// TwinCAT 3 PLC project TcoElements
// Title: TcoElements
// Company: Vortex.Library
// ProjectVersion: 0.6.0.913
// ProgramVersion: 3.1.4026.12
// libraries:
//   Tc2_Standard, * (Beckhoff Automation GmbH)
//   Tc2_System, * (Beckhoff Automation GmbH)
//   Tc3_Module, * (Beckhoff Automation GmbH)
//   TcoCore, 0.6.0.913 (Vortex.Library)
//   TcoUtilities, 0.6.0.913 (Vortex.Library)
// project tree:
//   Analog/TcoAi/ TcoAiAny.TcPOU (not stored), TcoAi.TcPOU (not stored), TcoAiConfig.TcDUT (not stored), TcoAiStatus.TcDUT (not stored)
//   Analog/TcoAo/ TcoAoConfig.TcDUT (not stored), TcoAoStatus.TcDUT (not stored), TcoAo.TcPOU (not stored)
//   Carousel/Base/ TcoCarouselBase.TcPOU (not stored)
//   Carousel/Structs/ eTcoCarouselDirection.TcDUT (not stored), TcoCarouselConfig.TcDUT (not stored), TcoCarouselStatus.TcDUT (not stored)
//   Carousel/Tasks/ TcoTurnTableTask.TcPOU (not stored)
//   Carousel/ TcoCarousel.TcPOU
//   Digital/TcoDi/ TcoDi.TcPOU, TcoDiConfig.TcDUT
//   Digital/TcoDo/ TcoDo.TcPOU
//   / PlcTask.TcTTO (not stored)
//   POUs/ MAIN.TcPOU (not stored)
// real-time tasks:
//   TASK PlcTask: cycle T#10ms, priority 20, ADS port 350
//   TASK PlcTask1: cycle T#10ms, priority 21, ADS port 351

// ---- Digital/TcoDi/TcoDiConfig.TcDUT
TYPE TcoDiConfig :
STRUCT
	IsFalseTimeOut : TIME := T#10S;
	IsTrueTimeOut : TIME := T#10S;
END_STRUCT
END_TYPE

// ---- Carousel/TcoCarousel.TcPOU
{attribute addProperty _turnTableName "<#Turn#>"}
{attribute addProperty _restoreName "<#Restore#>"}
FUNCTION_BLOCK TcoCarousel EXTENDS TcoCarouselBase
VAR_INPUT
		(*~
		<docu>
			<summary>
				This condition prevents the rotation of the table, possibly due to collisions with cylinders, axes, or other objects.
				Do not use signal from Light Curtain here.
			</summary>	
		</docu>
	~*)
	inSafetyCondition:BOOL;
	(*~
		<docu>
			<summary>
				The coded bites are stored in this word, which is valid for the base position of the carousel.
			</summary>	
		</docu>
	~*)
	inBasePositionNumber:WORD;
	
END_VAR
VAR
    {attribute addProperty Name "|[[1]Attribute_turnTableName]|"}
    _turnTask : TcoTurnTableTask(THIS^);

    {attribute addProperty Name "|[[1]Attribute_restoreName]|"}
    _restoreTask : TcoCore.TcoTask(THIS^);
    {attribute addProperty Name "<#Config#>"}
	_config : TcoCarouselConfig;
	{attribute addProperty Name "<#Status#>"}
	_status : TcoCarouselStatus;
END_VAR
VAR	
	increment: INT;
	_index: INT;	
	{attribute 'hide'}
	_positionsIdentifiersClear : ARRAY[0..20] OF UINT;

	_sb : TcoCore.StringBuilder;
	_basePositionNumber: WORD;
END_VAR

SUPER^( inoInPosition := inoInPosition, inoInPrecisePosition := inoInPrecisePosition, inoEnableTurn := inoEnableTurn, inoStartTurn := inoStartTurn);

_status.CurrentPosition:=	inBasePositionNumber;
_status.InPosition:=_inPosition;
_status.InPrecisePosition:=_inPrecisePosition;
_status.TurnSafetyCondition:=inSafetyCondition;




IF(_config.NumberOfPositions <= 0) THEN
	Messenger.Programming('- <#Parameter number of positions is <= 0. The paremeters must be grater than 0.#>'); 
	RETURN;
END_IF

_status.Positions :=_positionsIdentifiersClear;


IF(_config.OffSet = 0) THEN
	_config.OffSet := 1;
END_IF



// Calc position


_status.Positions[_config.NumberOfPositions - 1] := 1+(1 - _config.Offset + _status.CurrentPosition) MOD _config.NumberOfPositions;
FOR _index := 1 TO UINT_TO_INT(_config.NumberOfPositions) - 1 DO	
	_status.Positions[UINT_TO_INT(_config.NumberOfPositions) - 1 - _index] := 1 + ((_status.Positions[UINT_TO_INT(_config.NumberOfPositions) - _index]) MOD (_config.NumberOfPositions));			
END_FOR



// Disables mutualy exclusive actions		
_turnTask.Enabled := NOT _restoreTask.Busy;
	
_turnTask(
	inSafetyCondition:=inSafetyCondition , 
	inoInPosition:=_inPosition , 
	inoInPrecisePosition:=_inPrecisePosition , 
	inoEnableTurn:=_enableTurn , 
	inoStartTurn:=_startTurn , 
	inoConfig:=_config , 
	inoStatus:=_status );


_restoreTask.Enabled:=TRUE;

IF (_restoreTask.Execute()) THEN
 	Restore();

    _restoreTask.DoneWhen(TRUE);
END_IF

// For further discussion about Status
IF(_turnTask.Busy) THEN
	_status.ActionDescription := 'Roatating table to next position ';

ELSIF(_restoreTask.Busy) THEN
	_status.ActionDescription := 'Restoring';
ELSE	
	_status.ActionDescription := 'Idle';
END_IF

SUPER^(inoInPosition := inoInPosition, inoInPrecisePosition := inoInPrecisePosition, inoEnableTurn := inoEnableTurn, inoStartTurn := inoStartTurn);

(*~
	<docu>
		<summary>
			Aborts the turning when the condition is 'true'.
		</summary>
		<remarks>			
				<note type="warning">
					The call of this method will be effective only when called AFTER the initialization of the instance of given TcoCarousel.
				</note>
		</remarks>	
	</docu>
~*)
METHOD Abort : BOOL
VAR_IN_OUT
	(*~
		<docu>
			<summary>
				Condition to abort the turning of the carousel.
			</summary>	
		</docu>
	~*)
	inoDisableCondition : BOOL;
END_VAR
VAR_INPUT
	(*~
		<docu>
			<summary>
				Condition to abort the movement of the carousel can be inverted by this parameter.
			</summary>	
		</docu>
	~*)
	Invert:BOOL;
END_VAR
VAR
	_signalInfo : TcoSignalInfo;
END_VAR
IF ( _turnTask.Busy) AND inoDisableCondition AND NOT Invert THEN
	_signalInfo.GetSignalInfo(SIZEOF(inoDisableCondition), ADR(inoDisableCondition));
	Messenger.Build().Append('<#Turning table aborted due to#> : ').Append(_signalInfo.SymbolPath).As().AsError().Pin();
	_startTurn := FALSE;
	_enableTurn := FALSE;
	IF(__ISVALIDREF(THIS^.inoStartTurn)) THEN THIS^.inoStartTurn := FALSE; END_IF;
	IF(__ISVALIDREF(THIS^.inoEnableTurn)) THEN THIS^.inoEnableTurn := FALSE; END_IF;
	_turnTask.Abort();
ELSIF ( _turnTask.Busy) AND inoDisableCondition AND Invert THEN
	_signalInfo.GetSignalInfo(SIZEOF(inoDisableCondition), ADR(inoDisableCondition));
	Messenger.Build().Append('<#Turning table aborted due to NOT #> : ').Append(_signalInfo.SymbolPath).As().AsError().Pin();
	_startTurn := FALSE;
	_enableTurn := FALSE;
	IF(__ISVALIDREF(THIS^.inoStartTurn)) THEN THIS^.inoStartTurn := FALSE; END_IF;
	IF(__ISVALIDREF(THIS^.inoEnableTurn)) THEN THIS^.inoEnableTurn := FALSE; END_IF;
	_turnTask.Abort();
END_IF
END_METHOD

(*~
	<docu>
		<summary>
			Gets the `StopTask` task that controls the stopping the turning carousel. 		
		</summary>			
	</docu>	
~*)
PROPERTY AbortTask : TcoCore.ITcoTask
GET
AbortTask := _restoreTask;
END_GET
END_PROPERTY

PROPERTY Config : REFERENCE TO TcoCarouselConfig
GET
Config REF= _config;
END_GET
END_PROPERTY

METHOD PUBLIC GetIdentifierAtPosition : UINT
VAR_INPUT
	inPosition:UINT;
END_VAR
GetIdentifierAtPosition:=_turnTask.GetIdentifierAtPosition(inPosition:=inPosition,inPositions:=_status.Positions);
END_METHOD

(*~
	<docu>
		<summary>
			Restore all tasks of this instance into initial state.		 		 		
		</summary>			
	</docu>	
~*)
METHOD  Restore : ITcoRestorable
_turnTask.Restore();
_restoreTask.Abort();
_restoreTask.Restore();
_enableTurn := FALSE;
_startTurn := FALSE;
Messenger.UnPin();
END_METHOD

PROPERTY Status : REFERENCE TO TcoCarouselStatus
GET
Status REF= _status;
END_GET
END_PROPERTY

(*~
	<docu>
		<summary>
			Suspend the turning to next position when the condition is 'true'. Task is still bussy
		</summary>
		<remarks>			
				<note type="warning">
					The call of this method will be effective only when called AFTER the initialization of the instance of given TcoCarousel.
				</note>
		</remarks>	
	</docu>
~*)
METHOD Suspend : BOOL
VAR_IN_OUT
	(*~
		<docu>
			<summary>
				Condition to suspend the movement of the carousel.
			</summary>	
		</docu>
	~*)
	inoDisableCondition : BOOL;
END_VAR
VAR_INPUT
	(*~
		<docu>
			<summary>
				Condition to suspend the movement of the carousel can be inverted by this parameter.
			</summary>	
		</docu>
	~*)
	Invert:BOOL;
END_VAR
VAR
	_signalInfo : TcoSignalInfo;
END_VAR

IF (_turnTask.Busy OR _startTurn OR _enableTurn ) AND inoDisableCondition AND NOT Invert THEN
	_signalInfo.GetSignalInfo(SIZEOF(inoDisableCondition), ADR(inoDisableCondition));
	Messenger.Warning(_sb.Clear().Append('<#Turning table is suspended due to#> : ').Append(_signalInfo.SymbolPath).ToString());
	_startTurn := FALSE;
	_enableTurn := FALSE;
	IF(__ISVALIDREF(THIS^.inoStartTurn)) THEN THIS^.inoStartTurn := FALSE; END_IF;
	IF(__ISVALIDREF(THIS^.inoEnableTurn)) THEN THIS^.inoEnableTurn := FALSE; END_IF;
ELSIF (_turnTask.Busy OR _startTurn OR _enableTurn ) AND inoDisableCondition AND  Invert THEN
	_signalInfo.GetSignalInfo(SIZEOF(inoDisableCondition), ADR(inoDisableCondition));
	Messenger.Warning(_sb.Clear().Append('<#Turning table is suspended due to NOT #> : ').Append(_signalInfo.SymbolPath).ToString());
	_startTurn := FALSE;
	_enableTurn := FALSE;
	IF(__ISVALIDREF(THIS^.inoStartTurn)) THEN THIS^.inoStartTurn := FALSE; END_IF;
	IF(__ISVALIDREF(THIS^.inoEnableTurn)) THEN THIS^.inoEnableTurn := FALSE; END_IF;

END_IF
END_METHOD

METHOD SuspendExpression : BOOL
VAR_INPUT
		inDisableCondition : BOOL;
		inMessage:STRING;
END_VAR
IF (_turnTask.Busy OR _startTurn OR _enableTurn ) AND inDisableCondition THEN
	Messenger.Warning(CONCAT('<#Rotating is suspended due to#> : ' , inMessage));
	_startTurn := FALSE;
	_enableTurn := FALSE;
	IF(__ISVALIDREF(THIS^.inoStartTurn)) THEN THIS^.inoStartTurn := FALSE; END_IF;
	IF(__ISVALIDREF(THIS^.inoEnableTurn)) THEN THIS^.inoEnableTurn := FALSE; END_IF;
END_IF;
END_METHOD

(*~
	<docu>
		<summary>
			Gets the `TurnTask` task that controls the moving of the carousel to next position. 		
		</summary>			
	</docu>	
~*)
PROPERTY TurnTask : TcoCore.ITcoTask
GET
TurnTask := _turnTask;
END_GET
END_PROPERTY

END_FUNCTION_BLOCK

// ---- Digital/TcoDi/TcoDi.TcPOU
(*~
	<docu>
		<summary>
				Generic component for monitoring of an input. (e.g. DigitalSensor).												
		</summary>				
	</docu>	
~*)	
FUNCTION_BLOCK TcoDi EXTENDS TcoCore.TcoComponent
VAR_IN_OUT
	(*~
	<docu>
		<summary>
			Input signal. Typically an `%I*` variable. 												
		</summary>				
	</docu>	
	~*)
	inoSignal : BOOL;
END_VAR

VAR
	(*~
	<docu>
		<summary>
			Backing variable for signal; this variable is used directly by the component. It updates `inoSingal` in FB body call. 												
		</summary>				
	</docu>	
	~*)
	_signal : BOOL;	
END_VAR

VAR
	{attribute addProperty Name "<#Signal#>"}
	_signalInfo : TcoCore.TcoSignalInfo;
	{attribute addProperty Name "<#Check On#>"}
	{attribute addProperty ToolTip "<#Checks that the input is on#>"}
	_isTrueTask : TcoCore.TcoTask(THIS^);
	{attribute addProperty ToolTip "<#Checks that the input is off#>"}
	{attribute addProperty Name "<#Check Off#>"}
	_isFalseTask : TcoCore.TcoTask(THIS^);

	_config : TcoDiConfig;

	_isFalseTimeOutTimers : Tc2_Standard.TON;
	_isTrueTimeOutTimers : Tc2_Standard.TON;	
END_VAR

IF(__ISVALIDREF(inoSignal)) THEN
	_signalInfo.GetSignalInfo(SIZEOF(inoSignal), ADR(inoSignal));
	_signal := inoSignal;	
END_IF;	


IF(_isTrueTask.Execute())THEN
	_isTrueTask.DoneWhen(IsTrue);
END_IF

IF(_isFalseTask.Execute())THEN
	_isFalseTask.DoneWhen(IsFalse);
END_IF

PROPERTY Config : REFERENCE TO TcoDiConfig
GET
Config REF= _config;
END_GET
END_PROPERTY

METHOD FB_init : BOOL
VAR_INPUT
	bInitRetains : BOOL; // if TRUE, the retain variables are initialized (warm start / cold start)
	bInCopyCode : BOOL;  // if TRUE, the instance afterwards gets moved into the copy code (online change)
	ParentObject : ITcoObject;
END_VAR
END_METHOD

(*~
	<docu>
		<summary>
			Gets 'true' when monitor signal is 'off/false/logical 0'.
			Generates message when the returning 'false'.											
		</summary>				
	</docu>	
~*)	
{attribute 'monitoring' := 'variable'}
PROPERTY IsFalse : BOOL
GET
IsFalse := NOT _signal;
_isFalseTimeOutTimers(IN := NOT IsFalse, PT := _config.IsFalseTimeOut); 
IF(NOT IsFalse) THEN Messenger.Info('<#Expecting `negative` signal#>'); END_IF;
IF(_isFalseTimeOutTimers.Q) THEN Messenger.Warning('<#Expecting `negative` signal#>'); END_IF;
END_GET
END_PROPERTY

(*~
	<docu>
		<summary>
			Gets 'true' when monitor signal is 'on/true/logical 1'.
			Generates message when the returning 'false'.											
		</summary>				
	</docu>	
~*)	
{attribute 'monitoring' := 'variable'}
PROPERTY IsTrue : BOOL
GET
IsTrue := _signal;
_isTrueTimeOutTimers(IN := NOT IsTrue, PT := _config.IsFalseTimeOut); 
IF(NOT IsTrue) THEN Messenger.Info('<#Expecting `positive` signal#>'); END_IF;
IF(_isTrueTimeOutTimers.Q) THEN Messenger.Warning('<#Expecting `positive` signal#>'); END_IF;
END_GET
END_PROPERTY

(*~
	<docu>
		<summary>
			Restores this instance to the Ready state. Can be called explicitly or from within one of the restore mechanisms.	
		</summary>			
	</docu>	
~*)
METHOD  Restore : ITcoRestorable
// No implementation needed for this componet.
END_METHOD

(*~
	<docu>
		<summary>
		    Custom service (manual, maintenance) logic.
			This method must be implemented in derived class.
		</summary>			
	</docu>	
~*)
METHOD PROTECTED  ServiceMode
END_METHOD

PROPERTY PUBLIC Signal : Bool
GET
Signal :=  _signal;
END_GET
END_PROPERTY

END_FUNCTION_BLOCK

// ---- Digital/TcoDo/TcoDo.TcPOU
(*~
	<docu>
		<summary>
				Generic component for discrete control of an output.												
		</summary>				
	</docu>	
~*)
FUNCTION_BLOCK TcoDo EXTENDS TcoCore.TcoComponent
VAR_IN_OUT
	(*~
	<docu>
		<summary>
			Controlled signal. Typically an `%Q*` variable. 												
		</summary>				
	</docu>	
	~*)
	inoSignal : BOOL;
END_VAR

VAR
	(*~
	<docu>
		<summary>
			Backing variable for signal; this variable is used directly by the component. It updates `inoSingal` in FB body call. 												
		</summary>				
	</docu>	
	~*)
	_signal : BOOL;
END_VAR

VAR
	{attribute addProperty Name "<#Signal#>"}
	_signalInfo : TcoCore.TcoSignalInfo;
	{attribute addProperty Name "<#On#>"}
	{attribute addProperty ToolTip "<#Sets the output#>"}
	_setTask	 : TcoCore.TcoTask(THIS^);
	{attribute addProperty ToolTip "<#Resets the output#>"}
	{attribute addProperty Name "<#Off#>"}
	_resetTask	 : TcoCore.TcoTask(THIS^);
END_VAR

IF(__ISVALIDREF(inoSignal)) THEN
	_signalInfo.GetSignalInfo(SIZEOF(inoSignal), ADR(inoSignal));
	inoSignal := _signal;		 
END_IF;	
	
IF(_setTask.Execute())THEN
	_setTask.DoneWhen(Set());
END_IF

IF(_resetTask.Execute())THEN
	_resetTask.DoneWhen(Reset());
END_IF

METHOD FB_init : BOOL
VAR_INPUT
	bInitRetains : BOOL; // if TRUE, the retain variables are initialized (warm start / cold start)
	bInCopyCode : BOOL;  // if TRUE, the instance afterwards gets moved into the copy code (online change)
	ParentObject : ITcoObject;
END_VAR
END_METHOD

(*~
	<docu>
		<summary>
			Gets 'true' when monitor signal is 'off/false/logical 0'.
			Generates message when the returning 'false'.											
		</summary>				
	</docu>	
~*)	
{attribute 'monitoring' := 'variable'}
PROPERTY IsFalse : BOOL
GET
IsFalse := NOT _signal;
IF(NOT IsFalse) THEN Messenger.Info('<#Expecting `negative` signal#>'); END_IF;
END_GET
END_PROPERTY

(*~
	<docu>
		<summary>
			Gets 'true' when monitor signal is 'on/true/logical 1'.
			Generates message when the returning 'false'.											
		</summary>				
	</docu>	
~*)	
{attribute 'monitoring' := 'variable'}
PROPERTY IsTrue : BOOL
GET
IsTrue := _signal;
IF(NOT IsTrue) THEN Messenger.Info('<#Expecting `positive` signal#>'); END_IF;
END_GET
END_PROPERTY

(*~
	<docu>
		<summary>
			Sets controlled signal into 'off/false/logical 0'.														
		</summary>				
	</docu>	
~*)	
METHOD Reset : BOOL
Messenger.Trace('<#Reseting signal (off/false)#>');
_signal := FALSE;
Reset := TRUE;
END_METHOD

(*~
	<docu>
		<summary>
			Restores this instance to the Ready state. Can be called explicitly or from within one of the restore mechanisms.	
		</summary>			
	</docu>	
~*)
METHOD  Restore : ITcoRestorable
// No implementation needed for this componet.
END_METHOD

(*~
	<docu>
		<summary>
		    Custom service (manual, maintenance) logic.
			This method must be implemented in derived class.
		</summary>			
	</docu>	
~*)
METHOD PROTECTED  ServiceMode
END_METHOD

(*~
	<docu>
		<summary>
			Sets controlled signal into 'on/true/logical 1'.														
		</summary>				
	</docu>	
~*)	
METHOD PUBLIC Set : BOOL
Messenger.Trace('<#Setting signal (on/true)#>');
_signal := TRUE;
Set := TRUE;
END_METHOD

PROPERTY PUBLIC Signal : Bool
GET
Signal :=  _signal;
END_GET
END_PROPERTY

END_FUNCTION_BLOCK
